// TIA Portal V16 export
// export: Created 2021-11-12T13:32:33.2760587Z, ExportSetting WithDefaults, DisplayName Totally Integrated Automation Portal, DisplayVersion V16 Update 3, DisplayName TIA Portal Version Control Interface, DisplayVersion V16 Update 2, DisplayName TIA Portal Openness, DisplayVersion V16 Update 3, DisplayName SINAMICS Startdrive Advanced, DisplayVersion V16 Update 5, DisplayName SINAMICS Startdrive G130, G150, S120, S150, SINAMICS MV, S210, DisplayVersion V16 Update 5, DisplayName SINAMICS Startdrive G110M, G120, G120C, G120D, G120P, G115D, DisplayVersion V16 Update 5, DisplayName STEP 7 Professional, DisplayVersion V16 Update 3, DisplayName STEP 7 Safety, DisplayVersion V16, DisplayName WinCC UA Professional, DisplayVersion V16 Update 3
DATA_BLOCK "STATUS_Zone100"   // DB22
{ S7_Optimized_Access := 'TRUE'; DB_Accessible_From_OPC_UA := 'FALSE' }
VERSION : 0.1
// stored: AutoNumber true, DBAccessibleFromOPCUA false, IsOnlyStoredInLoadMemory false, IsRetainMemResEnabled false, IsWriteProtectedInAS false, MemoryReserve 100
   VAR
      Mode : Struct   // Status of zone 100
         Main : "UDT_Status_main";
         Specific : "UDT_Zone_Status_specific";
         Error : "UDT_Error01";
      END_STRUCT;
      StationKAS1_Mode : Struct   // Status of station saw KAS1
         Main : "UDT_Status_main";
         Specific : "UDT_Zone_Status_specific";
         Error : "UDT_Error01";
      END_STRUCT;
      StationKAS2_Mode : Struct   // Status of station saw KAS2
         Main : "UDT_Status_main";
         Specific : "UDT_Zone_Status_specific";
         Error : "UDT_Error01";
      END_STRUCT;
      Station110_Mode : Struct   // Status of station 110
         Main : "UDT_Status_main";
         Specific : "UDT_Zone_Status_specific";
         Error : "UDT_Error01";
      END_STRUCT;
      Station120_Mode : Struct   // Status of station 120
         Main : "UDT_Status_main";
         Specific : "UDT_Zone_Status_specific";
         Error : "UDT_Error01";
      END_STRUCT;
      Station1R1_Mode : Struct   // Status of station 1R1
         Main : "UDT_Status_main";
         Specific : "UDT_Zone_Status_specific";
         Error : "UDT_Error01";
      END_STRUCT;
      Station1R2_Mode : Struct   // Status of station 1R2
         Main : "UDT_Status_main";
         Specific : "UDT_Zone_Status_specific";
         Error : "UDT_Error01";
      END_STRUCT;
      Station130_Mode : Struct   // Status of station 130
         Main : "UDT_Status_main";
         Specific : "UDT_Zone_Status_specific";
         Error : "UDT_Error01";
      END_STRUCT;
      Station140_Mode : Struct   // Status of station 140
         Main : "UDT_Status_main";
         Specific : "UDT_Zone_Status_specific";
         Error : "UDT_Error01";
      END_STRUCT;
      Station1R3_Mode : Struct   // Status of station 1R3
         Main : "UDT_Status_main";
         Specific : "UDT_Zone_Status_specific";
         Error : "UDT_Error01";
      END_STRUCT;
      Station1R4_Mode : Struct   // Status of station 1R4
         Main : "UDT_Status_main";
         Specific : "UDT_Zone_Status_specific";
         Error : "UDT_Error01";
      END_STRUCT;
      Station150_Mode : Struct   // Status of station 150
         Main : "UDT_Status_main";
         Specific : "UDT_Zone_Status_specific";
         Error : "UDT_Error01";
      END_STRUCT;
      Station160_Mode : Struct   // Status of station 160
         Main : "UDT_Status_main";
         Specific : "UDT_Zone_Status_specific";
         Error : "UDT_Error01";
      END_STRUCT;
      Station170_Mode : Struct   // Status of station 170
         Main : "UDT_Status_main";
         Specific : "UDT_Zone_Status_specific";
         Error : "UDT_Error01";
      END_STRUCT;
      Station180_Mode : Struct   // Status of station 180
         Main : "UDT_Status_main";
         Specific : "UDT_Zone_Status_specific";
         Error : "UDT_Error01";
      END_STRUCT;
      Station1R5_Mode : Struct   // Status of station 1R5
         Main : "UDT_Status_main";
         Specific : "UDT_Zone_Status_specific";
         Error : "UDT_Error01";
      END_STRUCT;
      Station1R6_Mode : Struct   // Status of station 1R6
         Main : "UDT_Status_main";
         Specific : "UDT_Zone_Status_specific";
         Error : "UDT_Error01";
      END_STRUCT;
      StationBSN1_Mode : Struct   // Status of station furnace BSN1
         Main : "UDT_Status_main";
         Specific : "UDT_Zone_Status_specific";
         Error : "UDT_Error01";
      END_STRUCT;
      StationBSN2_Mode : Struct   // Status of station furnace BSN2
         Main : "UDT_Status_main";
         Specific : "UDT_Zone_Status_specific";
         Error : "UDT_Error01";
      END_STRUCT;
      "RU01-KF01" : Struct   // Status of bus module RU01-KF01
         Main : "UDT_Status_main";
         Specific { S7_SetPoint := 'True'} : "UDT_EuchnerSafetySwitch2MBM_Status_Specific";
         Error { S7_SetPoint := 'True'} : "UDT_Error01";
      END_STRUCT;
      "RU01-KF02" : Struct   // Status of bus module RU01-KF01
         Main : "UDT_Status_main";
         Specific { S7_SetPoint := 'True'} : "UDT_EuchnerSafetySwitch2MBM_Status_Specific";
         Error { S7_SetPoint := 'True'} : "UDT_Error01";
      END_STRUCT;
      "RU01-KF03" : Struct   // Status of bus module RU01-KF01
         Main : "UDT_Status_main";
         Specific { S7_SetPoint := 'True'} : "UDT_EuchnerSafetySwitch2MBM_Status_Specific";
         Error { S7_SetPoint := 'True'} : "UDT_Error01";
      END_STRUCT;
      "RU01-QQ01" : Struct   // Status of gate RU01-QQ01
         Main : "UDT_Status_main";
         Specific { S7_SetPoint := 'True'} : "UDT_Door_MGB2_L1_Status_specific";
         Error { S7_SetPoint := 'True'} : "UDT_Error01";
      END_STRUCT;
      "RU01-QQ02" : Struct   // Status of gate RU01-QQ02
         Main : "UDT_Status_main";
         Specific { S7_SetPoint := 'True'} : "UDT_Door_MGB2_L1_Status_specific";
         Error { S7_SetPoint := 'True'} : "UDT_Error01";
      END_STRUCT;
      "RU01-QQ03" : Struct   // Status of gate RU01-QQ03
         Main : "UDT_Status_main";
         Specific { S7_SetPoint := 'True'} : "UDT_Door_MGB2_L1_Status_specific";
         Error { S7_SetPoint := 'True'} : "UDT_Error01";
      END_STRUCT;
      "RU01-QQ04" : Struct   // Status of gate RU01-QQ04
         Main : "UDT_Status_main";
         Specific { S7_SetPoint := 'True'} : "UDT_Door_MGB2_L1_Status_specific";
         Error { S7_SetPoint := 'True'} : "UDT_Error01";
      END_STRUCT;
      "RU01-QQ05" : Struct   // Status of gate RU01-QQ05
         Main : "UDT_Status_main";
         Specific { S7_SetPoint := 'True'} : "UDT_Door_MGB2_L1_Status_specific";
         Error { S7_SetPoint := 'True'} : "UDT_Error01";
      END_STRUCT;
      "RU01-QQ06" : Struct   // Status of gate RU01-QQ06
         Main : "UDT_Status_main";
         Specific { S7_SetPoint := 'True'} : "UDT_Door_MGB2_L1_Status_specific";
         Error { S7_SetPoint := 'True'} : "UDT_Error01";
      END_STRUCT;
      "RU01-QQ07" : Struct   // Status of gate RU01-QQ07
         Main : "UDT_Status_main";
         Specific { S7_SetPoint := 'True'} : "UDT_Door_MGB2_L1_Status_specific";
         Error { S7_SetPoint := 'True'} : "UDT_Error01";
      END_STRUCT;
      "RU01-QQ08" : Struct   // Status of gate RU01-QQ08
         Main : "UDT_Status_main";
         Specific { S7_SetPoint := 'True'} : "UDT_Door_MGB2_L1_Status_specific";
         Error { S7_SetPoint := 'True'} : "UDT_Error01";
      END_STRUCT;
      xxxxx_Alarms__xxxxx : Byte;
      "UF01-SF01_ES" : Struct   // E-stop 100UF01-SF01
         Main { S7_SetPoint := 'True'} : "UDT_Status_main";
         Specific { S7_SetPoint := 'True'} : "UDT_DI_Mon_Status_specific";
         Error { S7_SetPoint := 'True'} : "UDT_Error01";
      END_STRUCT;
      "RU01-QQ01_ES" : Struct   // E-stop gate QQ01 / E-stop branka QQ01
         Main { S7_SetPoint := 'True'} : "UDT_Status_main";
         Specific { S7_SetPoint := 'True'} : "UDT_DI_Mon_Status_specific";
         Error { S7_SetPoint := 'True'} : "UDT_Error01";
      END_STRUCT;
      "RU01-QQ02_ES" : Struct   // E-stop gate QQ02 / E-stop branka QQ02
         Main { S7_SetPoint := 'True'} : "UDT_Status_main";
         Specific { S7_SetPoint := 'True'} : "UDT_DI_Mon_Status_specific";
         Error { S7_SetPoint := 'True'} : "UDT_Error01";
      END_STRUCT;
      "RU01-QQ03_ES" : Struct   // E-stop gate QQ03 / E-stop branka QQ03
         Main { S7_SetPoint := 'True'} : "UDT_Status_main";
         Specific { S7_SetPoint := 'True'} : "UDT_DI_Mon_Status_specific";
         Error { S7_SetPoint := 'True'} : "UDT_Error01";
      END_STRUCT;
      "RU01-QQ04_ES" : Struct   // E-stop gate QQ04 / E-stop branka QQ04
         Main { S7_SetPoint := 'True'} : "UDT_Status_main";
         Specific { S7_SetPoint := 'True'} : "UDT_DI_Mon_Status_specific";
         Error { S7_SetPoint := 'True'} : "UDT_Error01";
      END_STRUCT;
      "RU01-QQ05_ES" : Struct   // E-stop gate QQ05 / E-stop branka QQ05
         Main { S7_SetPoint := 'True'} : "UDT_Status_main";
         Specific { S7_SetPoint := 'True'} : "UDT_DI_Mon_Status_specific";
         Error { S7_SetPoint := 'True'} : "UDT_Error01";
      END_STRUCT;
      "RU01-QQ06_ES" : Struct   // E-stop gate QQ06 / E-stop branka QQ06
         Main { S7_SetPoint := 'True'} : "UDT_Status_main";
         Specific { S7_SetPoint := 'True'} : "UDT_DI_Mon_Status_specific";
         Error { S7_SetPoint := 'True'} : "UDT_Error01";
      END_STRUCT;
      "RU01-QQ07_ES" : Struct   // E-stop gate QQ07 / E-stop branka QQ07
         Main { S7_SetPoint := 'True'} : "UDT_Status_main";
         Specific { S7_SetPoint := 'True'} : "UDT_DI_Mon_Status_specific";
         Error { S7_SetPoint := 'True'} : "UDT_Error01";
      END_STRUCT;
      "RU01-QQ08_ES" : Struct   // E-stop gate QQ08 / E-stop branka QQ08
         Main { S7_SetPoint := 'True'} : "UDT_Status_main";
         Specific { S7_SetPoint := 'True'} : "UDT_DI_Mon_Status_specific";
         Error { S7_SetPoint := 'True'} : "UDT_Error01";
      END_STRUCT;
      "RU01-KF2" : Struct   // gate module 100RU01-KF01
         Main { S7_SetPoint := 'True'} : "UDT_Status_main";
         Specific { S7_SetPoint := 'True'} : "UDT_DI_Mon_Status_specific";
         Error { S7_SetPoint := 'True'} : "UDT_Error01";
      END_STRUCT;
      "RU01-KF3" : Struct   // gate module 100RU01-KF02
         Main { S7_SetPoint := 'True'} : "UDT_Status_main";
         Specific { S7_SetPoint := 'True'} : "UDT_DI_Mon_Status_specific";
         Error { S7_SetPoint := 'True'} : "UDT_Error01";
      END_STRUCT;
      "RU01-KF4" : Struct   // gate module 100RU01-KF03
         Main { S7_SetPoint := 'True'} : "UDT_Status_main";
         Specific { S7_SetPoint := 'True'} : "UDT_DI_Mon_Status_specific";
         Error { S7_SetPoint := 'True'} : "UDT_Error01";
      END_STRUCT;
      ChangeToolNotDone : Struct
         "1R1" : Bool;   // 1R1 has not finished changing tool process / 1R1 nedokončený proces výměny nástrojů
         "1R2" : Bool;   // 1R2 has not finished changing tool process / 1R2 nedokončený proces výměny nástrojů
         "1R3" : Bool;   // 1R3 has not finished changing tool process / 1R3 nedokončený proces výměny nástrojů
         "1R4" : Bool;   // 1R4 has not finished changing tool process / 1R4 nedokončený proces výměny nástrojů
         "1R5" : Bool;   // 1R5 has not finished changing tool process / 1R5 nedokončený proces výměny nástrojů
         "1R6" : Bool;   // 1R6 has not finished changing tool process / 1R6 nedokončený proces výměny nástrojů
      END_STRUCT;
   END_VAR
BEGIN
END_DATA_BLOCK
